Staubli VAL3: Body.dtx

public num nData
